INTERFACE I_MotionLogger

END_INTERFACE

(* stored: Version 1.1.0.1
   Itf I_MotionLogger: Id {ba839cec-9291-4692-8f1c-76e0f27d3db4} *)
